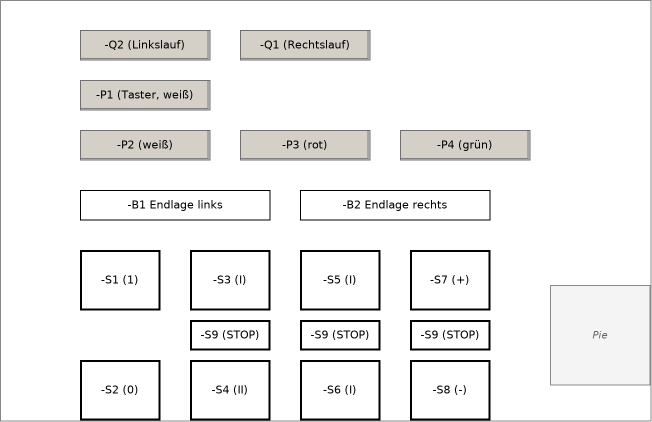
VISUALIZATION WordClock  // 652x422
    Button (80,80 130x30), "-P1 (Taster, weiß)"
        tap dSub.P1
    Button (80,130 130x30), "-P2 (weiß)"
        tap dSub.P2
    Button (240,130 130x30), "-P3 (rot)"
        tap dSub.P3
    Button (400,130 130x30), "-P4 (grün)"
        tap dSub.P4
    Button (240,30 130x30), "-Q1 (Rechtslauf)"
        tap dSub.Q1
    Button (80,30 130x30), "-Q2 (Linkslauf)"
        tap dSub.Q2
    Rectangle (80,250 80x60), "-S1 (1)", colour toggle: dSub.S1
    Rectangle (80,360 80x60), "-S2 (0)", colour toggle: dSub.S2
    Rectangle (190,250 80x60), "-S3 (I)", colour toggle: dSub.S3
    Rectangle (190,360 80x60), "-S4 (II)", colour toggle: dSub.S4
    Rectangle (190,320 80x30), "-S9 (STOP)", colour toggle: dSub.S9
    Rectangle (300,250 80x60), "-S5 (I)", colour toggle: dSub.S5
    Rectangle (300,360 80x60), "-S6 (I)", colour toggle: dSub.S6
    Rectangle (300,320 80x30), "-S9 (STOP)", colour toggle: dSub.S9
    Rectangle (410,250 80x60), "-S7 (+)", colour toggle: dSub.S7
    Rectangle (410,360 80x60), "-S8 (-)", colour toggle: dSub.S8
    Rectangle (410,320 80x30), "-S9 (STOP)", colour toggle: dSub.S9
    Pie (550,285 100x100), colour toggle: dSub.S11
    Pie (550,285 100x100), colour toggle: dSub.S10
    Rectangle (80,190 190x30), "-B1 Endlage links", colour toggle: dSub.B1
    Rectangle (300,190 190x30), "-B2 Endlage rechts", colour toggle: dSub.B2
END_VISUALIZATION

(* stored: Version 1.1.0.1, ProductVersion 3.1.4022.7
   Visu WordClock: Id {529ab607-a3a7-4016-be48-cafee3caa910} *)
